(* B8 = Reset *)
TYPE ST_B8Res :
STRUCT
	PathID			:UINT;		(* 2 bytes*)
	CRC1			:BYTE;	    (* 1 byte*)
	CRC2			:BYTE;	    (* 1 byte*)			
END_STRUCT
END_TYPE

(* stored: Version 1.1.0.1, ProductVersion 3.1.4020.12
   DUT ST_B8Res: Id {03778315-288d-4584-b9fa-a47576c796ae} *)
